(* PLC project Unnamed, Unknown Unnamed 1 *)
(* stored: creationDateTime 2025-02-04T11:16:08, modificationDateTime 2025-02-05T14:31:39 *)

(* Copy type A parameters from input to output *)
FUNCTION_BLOCK move_A
  VAR_IN_OUT
    Product_Name : STRING;
    Product_Image : INT;
    Step_1_Bake_Time : DINT;
    Step_1_Bake_Temp : DINT;
    Step_2_Bake_Time : DINT;
    Step_2_Bake_Temp : DINT;
  END_VAR

            (* Nothing to do here *)
RETURN;

          
END_FUNCTION_BLOCK

FUNCTION_BLOCK machine_A
  VAR_INPUT
    Step_1_Bake_Time : DINT;
    Step_1_Bake_Temp : DINT;
    Step_2_Bake_Time : DINT;
    Step_2_Bake_Temp : DINT;
  END_VAR
  VAR
    local_dint : DINT;
  END_VAR

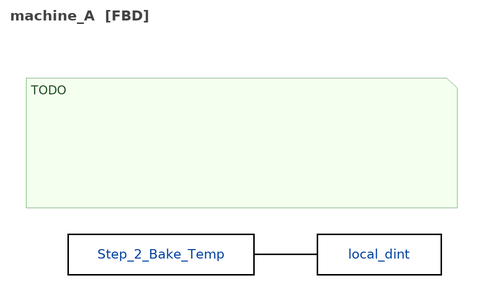
(* FBD diagram, written out as Structured Text *)
(* TODO *)
local_dint := Step_2_Bake_Temp;
END_FUNCTION_BLOCK

(* Read CSV file of type A *)
FUNCTION_BLOCK write_csv_A
  VAR_INPUT
    CSV_NAME : STRING;  (* CSV file name *)
    SAVE : BOOL;  (* Triggers CSV file read on rising edge *)
  END_VAR
  VAR_OUTPUT
    ERROR : BOOL;  (* Write operation failed *)
    ACK : BOOL;  (* Output is valid *)
  END_VAR
  VAR_INPUT
    Product_Name : STRING;
    Product_Image : INT;
    Step_1_Bake_Time : DINT;
    Step_1_Bake_Temp : DINT;
    Step_2_Bake_Time : DINT;
    Step_2_Bake_Temp : DINT;
  END_VAR
  VAR
    csv_write_by_string0 : csv_write_by_string;
    csv_write_by_string1 : csv_write_by_string;
    csv_write_by_string2 : csv_write_by_string;
    csv_write_by_string3 : csv_write_by_string;
    csv_write_by_string4 : csv_write_by_string;
    csv_write_by_string5 : csv_write_by_string;
  END_VAR

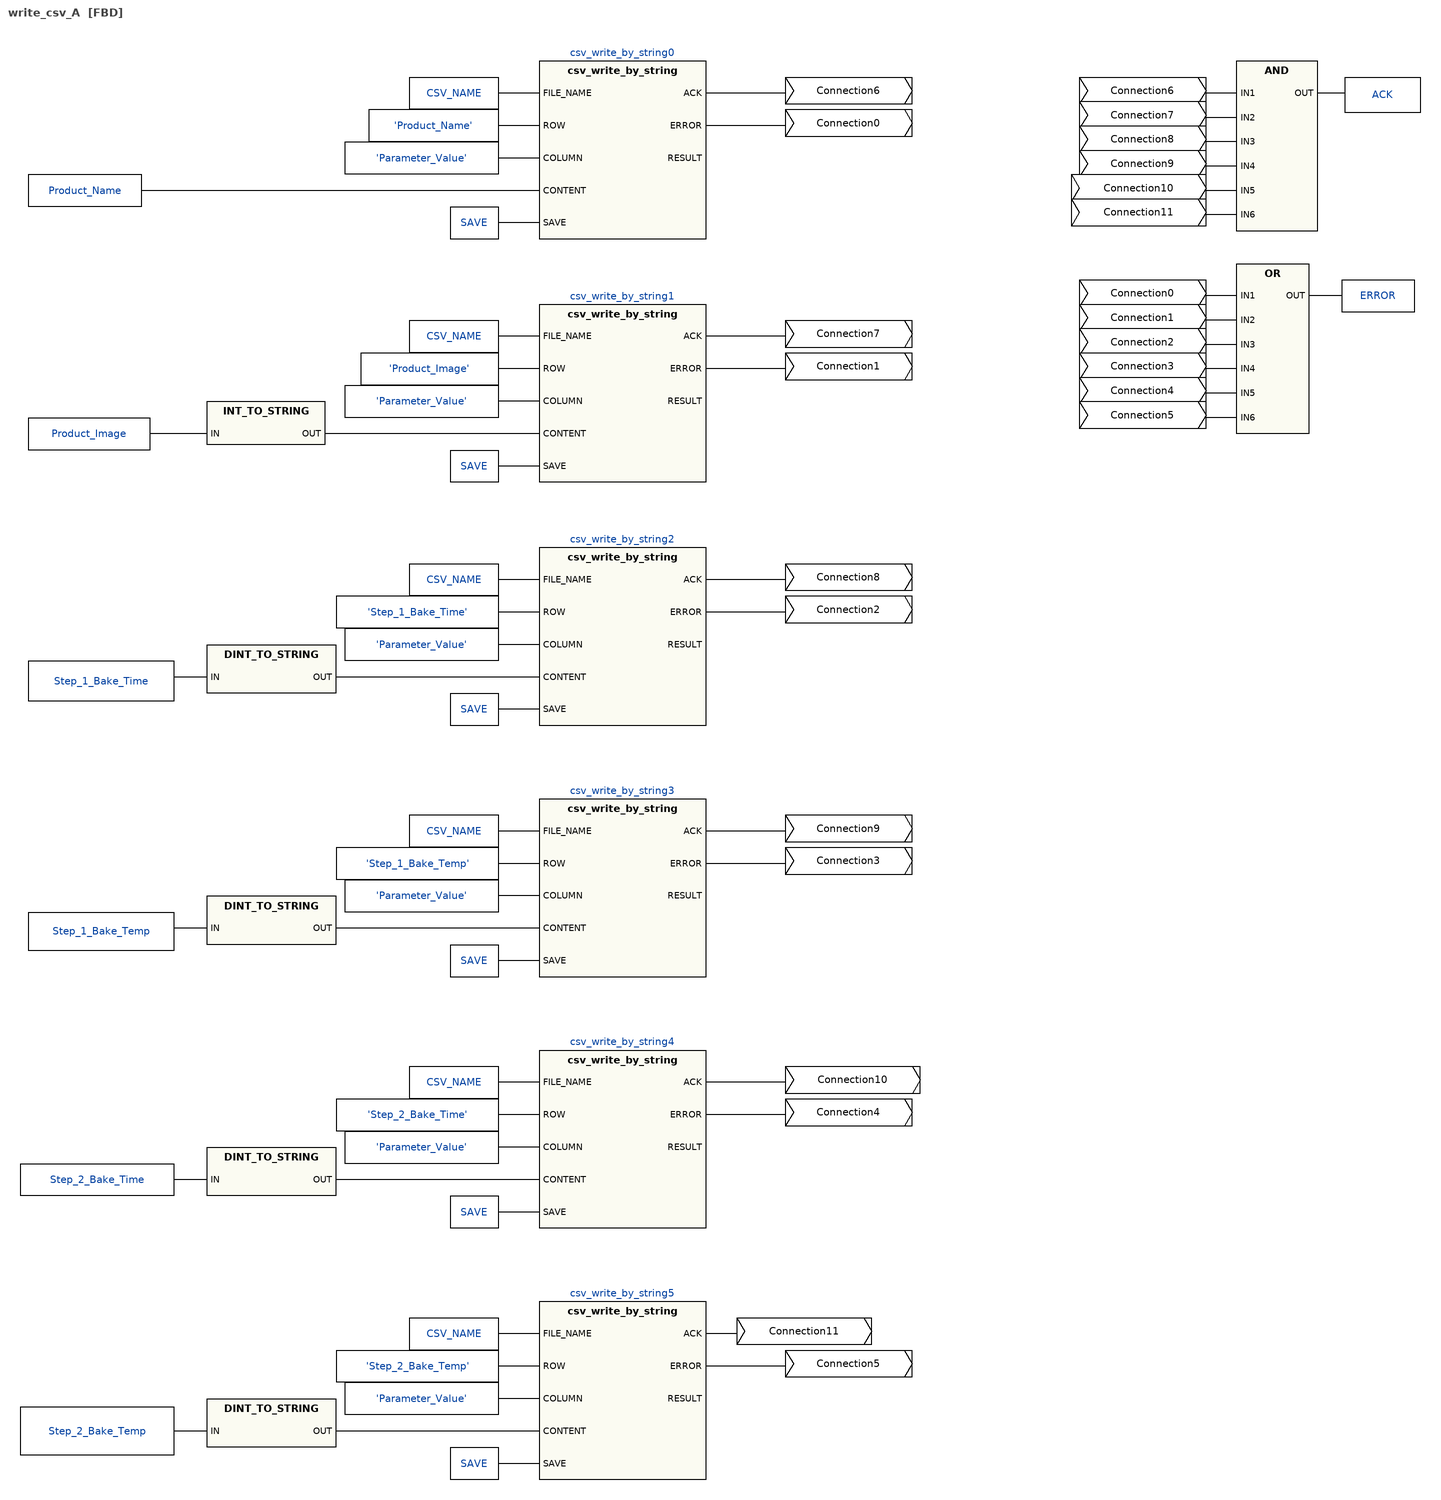
(* FBD diagram, written out as Structured Text *)
csv_write_by_string0(FILE_NAME := CSV_NAME, ROW := 'Product_Name', COLUMN := 'Parameter_Value', CONTENT := Product_Name, SAVE := SAVE);
csv_write_by_string1(FILE_NAME := CSV_NAME, ROW := 'Product_Image', COLUMN := 'Parameter_Value', CONTENT := INT_TO_STRING(Product_Image), SAVE := SAVE);
csv_write_by_string2(FILE_NAME := CSV_NAME, ROW := 'Step_1_Bake_Time', COLUMN := 'Parameter_Value', CONTENT := DINT_TO_STRING(Step_1_Bake_Time), SAVE := SAVE);
csv_write_by_string3(FILE_NAME := CSV_NAME, ROW := 'Step_1_Bake_Temp', COLUMN := 'Parameter_Value', CONTENT := DINT_TO_STRING(Step_1_Bake_Temp), SAVE := SAVE);
csv_write_by_string4(FILE_NAME := CSV_NAME, ROW := 'Step_2_Bake_Time', COLUMN := 'Parameter_Value', CONTENT := DINT_TO_STRING(Step_2_Bake_Time), SAVE := SAVE);
csv_write_by_string5(FILE_NAME := CSV_NAME, ROW := 'Step_2_Bake_Temp', COLUMN := 'Parameter_Value', CONTENT := DINT_TO_STRING(Step_2_Bake_Temp), SAVE := SAVE);
ERROR := csv_write_by_string0.ERROR OR csv_write_by_string1.ERROR OR csv_write_by_string2.ERROR OR csv_write_by_string3.ERROR OR csv_write_by_string4.ERROR OR csv_write_by_string5.ERROR;
ACK := csv_write_by_string0.ACK AND csv_write_by_string1.ACK AND csv_write_by_string2.ACK AND csv_write_by_string3.ACK AND csv_write_by_string4.ACK AND csv_write_by_string5.ACK;
END_FUNCTION_BLOCK

(* Read CSV file of type A *)
FUNCTION_BLOCK read_csv_A
  VAR_INPUT
    CSV_NAME : STRING;  (* CSV file name *)
  END_VAR
  VAR_OUTPUT
    SUCCESS : BOOL;  (* TRUE if data comes from file FALSE if default values *)
    Product_Name : STRING := 'unknown';
    Product_Image : INT := 0;
    Step_1_Bake_Time : DINT := 60;
    Step_1_Bake_Temp : DINT := 120;
    Step_2_Bake_Time : DINT := 90;
    Step_2_Bake_Temp : DINT := 180;
  END_VAR
  VAR
    csv_read_by_string0 : csv_read_by_string;
    csv_read_by_string1 : csv_read_by_string;
    csv_read_by_string2 : csv_read_by_string;
    csv_read_by_string3 : csv_read_by_string;
    csv_read_by_string4 : csv_read_by_string;
    csv_read_by_string5 : csv_read_by_string;
  END_VAR
  VAR  (* added by the conversion: wires and edge detectors of the diagram *)
    _STRING_TO_INT11_ENO : BOOL;
    _STRING_TO_INT11_OUT : INT;
    _STRING_TO_DINT17_ENO : BOOL;
    _STRING_TO_DINT17_OUT : DINT;
    _STRING_TO_DINT23_ENO : BOOL;
    _STRING_TO_DINT23_OUT : DINT;
    _STRING_TO_DINT29_ENO : BOOL;
    _STRING_TO_DINT29_OUT : DINT;
    _STRING_TO_DINT35_ENO : BOOL;
    _STRING_TO_DINT35_OUT : DINT;
  END_VAR

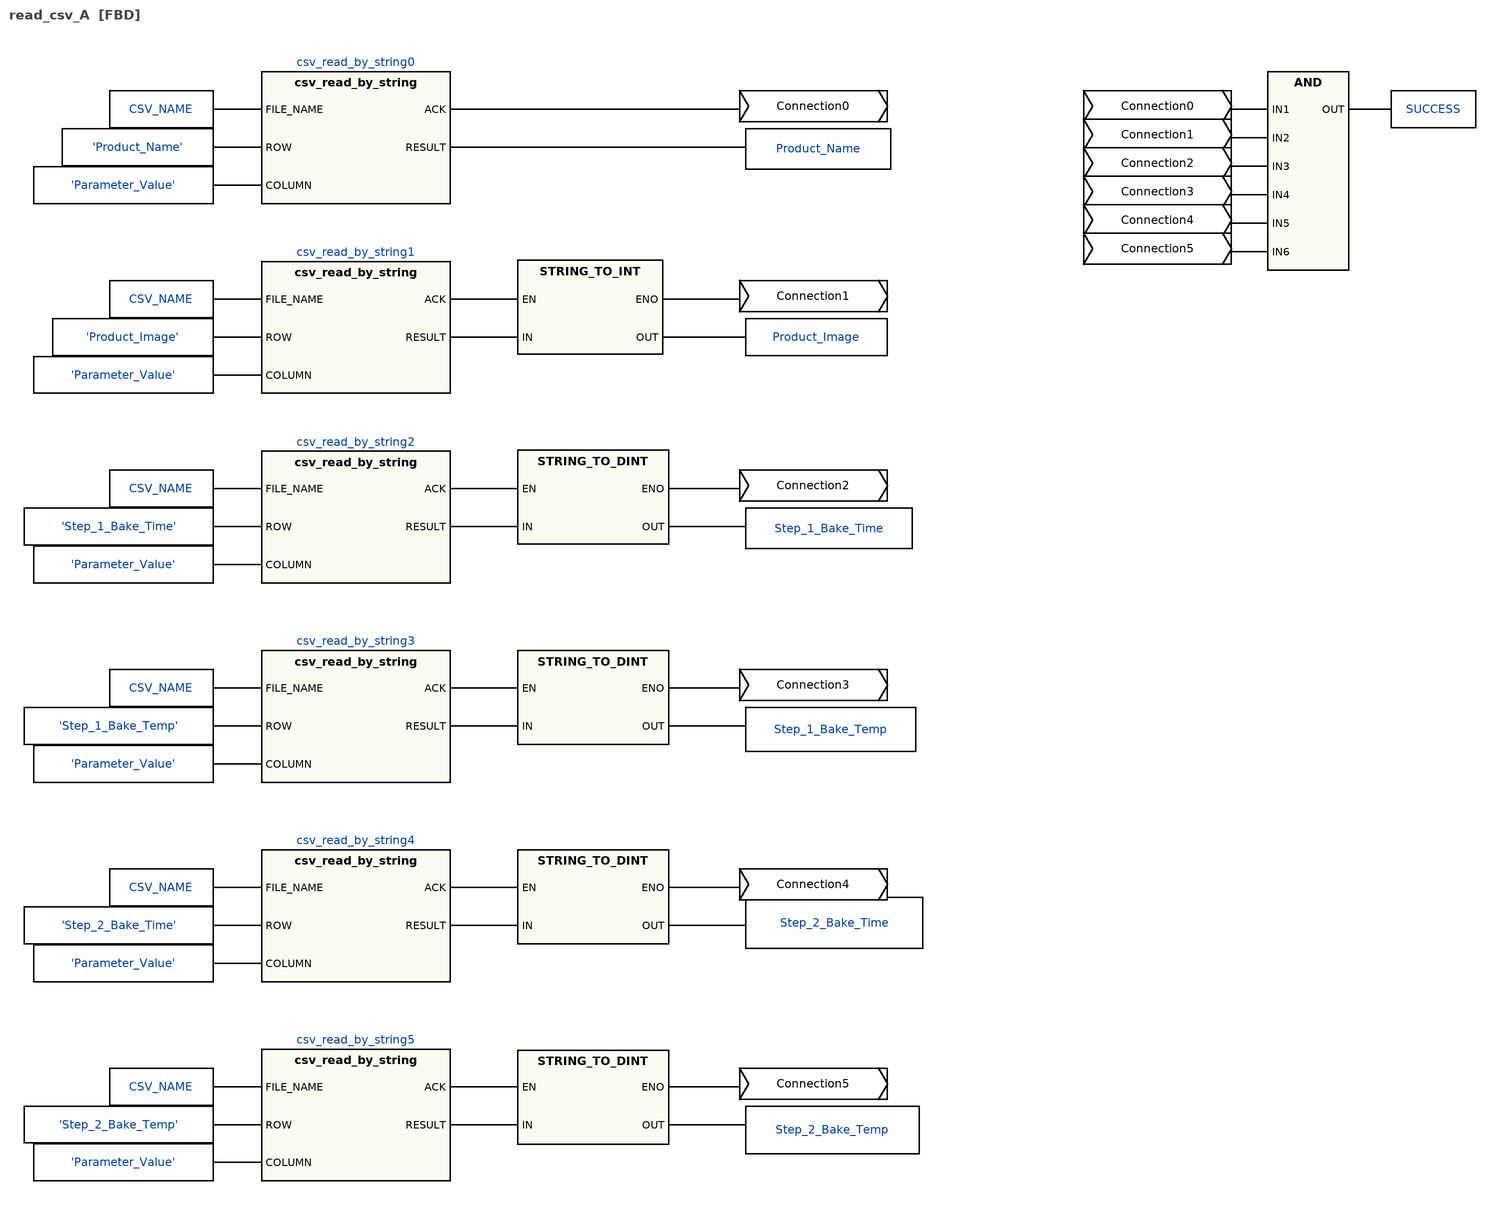
(* FBD diagram, written out as Structured Text *)
csv_read_by_string0(FILE_NAME := CSV_NAME, ROW := 'Product_Name', COLUMN := 'Parameter_Value');
Product_Name := csv_read_by_string0.RESULT;
csv_read_by_string1(FILE_NAME := CSV_NAME, ROW := 'Product_Image', COLUMN := 'Parameter_Value');
_STRING_TO_INT11_OUT := STRING_TO_INT(EN := csv_read_by_string1.ACK, IN := csv_read_by_string1.RESULT, ENO => _STRING_TO_INT11_ENO);
IF _STRING_TO_INT11_ENO THEN Product_Image := _STRING_TO_INT11_OUT; END_IF;
csv_read_by_string2(FILE_NAME := CSV_NAME, ROW := 'Step_1_Bake_Time', COLUMN := 'Parameter_Value');
_STRING_TO_DINT17_OUT := STRING_TO_DINT(EN := csv_read_by_string2.ACK, IN := csv_read_by_string2.RESULT, ENO => _STRING_TO_DINT17_ENO);
IF _STRING_TO_DINT17_ENO THEN Step_1_Bake_Time := _STRING_TO_DINT17_OUT; END_IF;
csv_read_by_string3(FILE_NAME := CSV_NAME, ROW := 'Step_1_Bake_Temp', COLUMN := 'Parameter_Value');
_STRING_TO_DINT23_OUT := STRING_TO_DINT(EN := csv_read_by_string3.ACK, IN := csv_read_by_string3.RESULT, ENO => _STRING_TO_DINT23_ENO);
IF _STRING_TO_DINT23_ENO THEN Step_1_Bake_Temp := _STRING_TO_DINT23_OUT; END_IF;
csv_read_by_string4(FILE_NAME := CSV_NAME, ROW := 'Step_2_Bake_Time', COLUMN := 'Parameter_Value');
_STRING_TO_DINT29_OUT := STRING_TO_DINT(EN := csv_read_by_string4.ACK, IN := csv_read_by_string4.RESULT, ENO => _STRING_TO_DINT29_ENO);
IF _STRING_TO_DINT29_ENO THEN Step_2_Bake_Time := _STRING_TO_DINT29_OUT; END_IF;
csv_read_by_string5(FILE_NAME := CSV_NAME, ROW := 'Step_2_Bake_Temp', COLUMN := 'Parameter_Value');
_STRING_TO_DINT35_OUT := STRING_TO_DINT(EN := csv_read_by_string5.ACK, IN := csv_read_by_string5.RESULT, ENO => _STRING_TO_DINT35_ENO);
IF _STRING_TO_DINT35_ENO THEN Step_2_Bake_Temp := _STRING_TO_DINT35_OUT; END_IF;
SUCCESS := csv_read_by_string0.ACK AND _STRING_TO_INT11_ENO AND _STRING_TO_DINT17_ENO AND _STRING_TO_DINT23_ENO AND _STRING_TO_DINT29_ENO AND _STRING_TO_DINT35_ENO;
END_FUNCTION_BLOCK

PROGRAM program0
  VAR
    SAVE_BT : HMI_BOOL;
    SAVE_AS_BT : HMI_BOOL;
    RD_SUCCESS : HMI_BOOL;
    SAVE_ACK : HMI_BOOL;
    SAVE_SUCCESS : HMI_BOOL;
    CURRENT_CSV : HMI_STRING := test.csv;
    SAVE_AS_CSV : HMI_STRING := test2.csv;
    Product_Name : HMI_STRING := 'unknown';
    Product_Image : HMI_INT := 0;
    Step_1_Bake_Time : HMI_DINT := 60;
    Step_1_Bake_Temp : HMI_DINT := 120;
    Step_2_Bake_Time : HMI_DINT := 90;
    Step_2_Bake_Temp : HMI_DINT := 180;
    read_csv_A0 : read_csv_A;
    write_csv_A0 : write_csv_A;
    machine_A0 : machine_A;
    move_A0 : move_A;
  END_VAR
  VAR  (* added by the conversion: wires and edge detectors of the diagram *)
    R_TRIG1 : R_TRIG;
  END_VAR

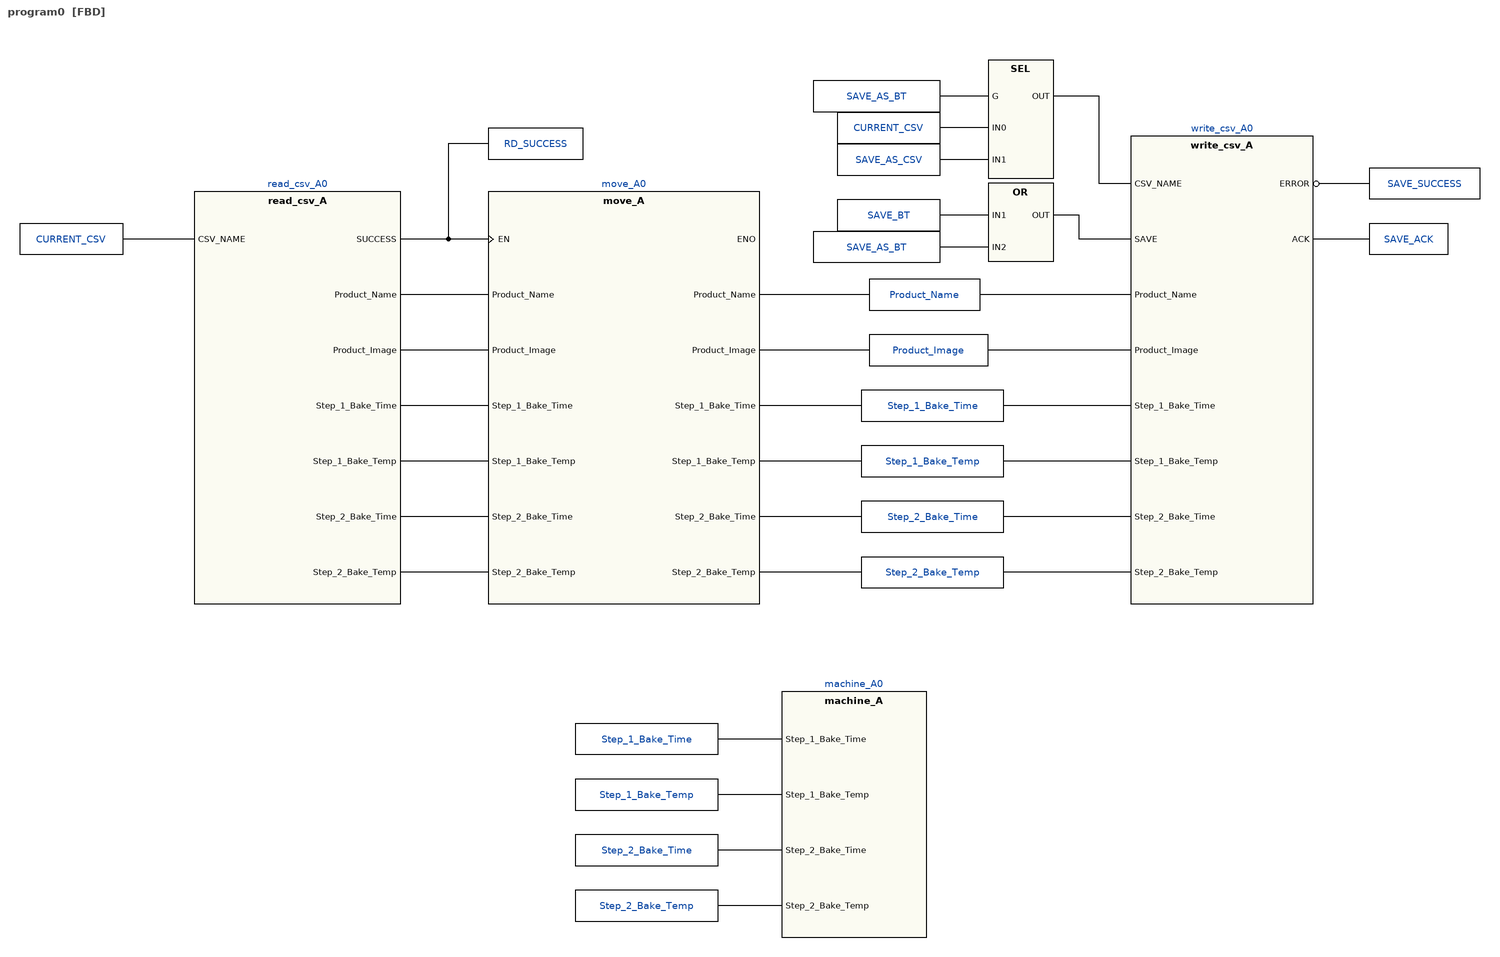
(* FBD diagram, written out as Structured Text *)
read_csv_A0(CSV_NAME := CURRENT_CSV);
R_TRIG1(CLK := read_csv_A0.SUCCESS);
move_A0(EN := R_TRIG1.Q, Product_Name := read_csv_A0.Product_Name, Product_Image := read_csv_A0.Product_Image, Step_1_Bake_Time := read_csv_A0.Step_1_Bake_Time, Step_1_Bake_Temp := read_csv_A0.Step_1_Bake_Temp, Step_2_Bake_Time := read_csv_A0.Step_2_Bake_Time, Step_2_Bake_Temp := read_csv_A0.Step_2_Bake_Temp);
IF move_A0.ENO THEN Product_Name := move_A0.Product_Name; END_IF;
IF move_A0.ENO THEN Product_Image := move_A0.Product_Image; END_IF;
IF move_A0.ENO THEN Step_1_Bake_Time := move_A0.Step_1_Bake_Time; END_IF;
IF move_A0.ENO THEN Step_1_Bake_Temp := move_A0.Step_1_Bake_Temp; END_IF;
IF move_A0.ENO THEN Step_2_Bake_Time := move_A0.Step_2_Bake_Time; END_IF;
IF move_A0.ENO THEN Step_2_Bake_Temp := move_A0.Step_2_Bake_Temp; END_IF;
RD_SUCCESS := read_csv_A0.SUCCESS;
write_csv_A0(CSV_NAME := SEL(SAVE_AS_BT, CURRENT_CSV, SAVE_AS_CSV), SAVE := SAVE_BT OR SAVE_AS_BT, Product_Name := Product_Name, Product_Image := Product_Image, Step_1_Bake_Time := Step_1_Bake_Time, Step_1_Bake_Temp := Step_1_Bake_Temp, Step_2_Bake_Time := Step_2_Bake_Time, Step_2_Bake_Temp := Step_2_Bake_Temp);
SAVE_SUCCESS := NOT write_csv_A0.ERROR;
SAVE_ACK := write_csv_A0.ACK;
machine_A0(Step_1_Bake_Time := Step_1_Bake_Time, Step_1_Bake_Temp := Step_1_Bake_Temp, Step_2_Bake_Time := Step_2_Bake_Time, Step_2_Bake_Temp := Step_2_Bake_Temp);
END_PROGRAM

CONFIGURATION config
  RESOURCE resource1 ON PLC
    TASK task0(INTERVAL := T#20ms, PRIORITY := 0);
    PROGRAM instance0 WITH task0 : program0;
  END_RESOURCE
END_CONFIGURATION
